// TIA Portal V16 program export: 2 tag tables, 0 data types, 2 data blocks, 14 code blocks (in call order from the OBs), 13 instance data blocks

VAR_GLOBAL   // PLC tag table "Default tag table"
   FIC_B102 AT %IW64 : Int;
   LIC_B101 AT %IW66 : Int;
   PS1_RFID_Station AT %I0.0 : Bool;   // PS-Proximity Switch
   PS2_Filling_Station AT %I0.1 : Bool;
   PS3_Quality_Station AT %I0.2 : Bool;
   PS4_End_of_Conveyor AT %I0.3 : Bool;
   T01_Low_Level AT %I0.4 : Bool;
   T01_High_Level AT %I0.5 : Bool;
   T01_Outlet AT %Q0.1 : Bool;
   T02_Outlet AT %Q0.2 : Bool;
   Outlet_Pump_Motor AT %Q0.3 : Bool;
   Conveyor_Motor AT %Q0.0 : Bool;
   NTRG_06 AT %M5.5 : Bool;
   NTRG_09 AT %M5.6 : Bool;
   NTRG_099 AT %M5.7 : Bool;
   PTRG10 AT %M6.0 : Bool;
   PTRIG999 AT %M6.1 : Bool;
   PTRIG998 AT %M6.2 : Bool;
   PTRIG888 AT %M6.3 : Bool;
   ptrig141 AT %M6.4 : Bool;
   ptrig142 AT %M6.5 : Bool;
   ptrig143 AT %M6.6 : Bool;
END_VAR

VAR_GLOBAL   // PLC tag table "P_N_TRIG"
   PTRIG1 AT %M0.0 : Bool;
   PTRIG2 AT %M0.1 : Bool;
   PTRIG3 AT %M0.2 : Bool;
   PTRIG4 AT %M0.3 : Bool;
   PTRIG5 AT %M0.4 : Bool;
   PTRIG6 AT %M0.5 : Bool;
   PTRIG7 AT %M0.6 : Bool;
   PTRIG8 AT %M0.7 : Bool;
   PTRIG9 AT %M1.0 : Bool;
   PTRIG10 AT %M1.1 : Bool;
   PTRIG11 AT %M1.2 : Bool;
   PTRIG12 AT %M1.3 : Bool;
   PTRIG13 AT %M1.4 : Bool;
   PTRIG14 AT %M1.5 : Bool;
   PTRIG15 AT %M1.6 : Bool;
   PTRIG16 AT %M1.7 : Bool;
   PTRIG17 AT %M2.0 : Bool;
   PTRIG18 AT %M2.1 : Bool;
   PTRIG19 AT %M2.2 : Bool;
   PTRIG20 AT %M2.3 : Bool;
   PTRIG21 AT %M2.4 : Bool;
   PTRIG22 AT %M2.5 : Bool;
   PTRIG23 AT %M2.6 : Bool;
   NTRIG1 AT %M2.7 : Bool;
   NTRIG2 AT %M3.0 : Bool;
   NTRIG3 AT %M3.1 : Bool;
   NTRIG4 AT %M3.2 : Bool;
   NTRIG5 AT %M3.3 : Bool;
   NTRIG6 AT %M3.4 : Bool;
   NTRIG7 AT %M3.5 : Bool;
   NTRIG8 AT %M3.6 : Bool;
   NTRIG9 AT %M3.7 : Bool;
   NTRIG10 AT %M4.0 : Bool;
   NTRIG11 AT %M4.1 : Bool;
   NTRIG12 AT %M4.2 : Bool;
   NTRIG13 AT %M4.3 : Bool;
   NTRIG14 AT %M4.4 : Bool;
   NTRIG15 AT %M4.5 : Bool;
   NTRIG16 AT %M4.6 : Bool;
   NTRIG17 AT %M4.7 : Bool;
   NTRIG18 AT %M5.0 : Bool;
   NTRIG19 AT %M5.1 : Bool;
   NTRIG20 AT %M5.2 : Bool;
   PTRIG24 AT %M5.3 : Bool;
   PTRIG25 AT %M5.4 : Bool;
END_VAR

DATA_BLOCK "DuplicateDB"   // DB12
{ S7_Optimized_Access := 'FALSE' }
VERSION : 0.1
// stored: AutoNumber true, DBAccessibleFromOPCUA true, IsOnlyStoredInLoadMemory false, IsWriteProtectedInAS false
   VAR
      Input : Struct
         FIC_B102 : Int;   // Tank2 Level Measurement
         LIC_B101 : Int;
         PS1_RFID_Station : Bool;
         PS2_Filling_Station : Bool;
         PS3_Quality_Station : Bool;
         PS4_End_of_Conveyor : Bool;
         T01_Low_Level : Bool;
         T01_High_Level : Bool;
      END_STRUCT;
   END_VAR
BEGIN
END_DATA_BLOCK

DATA_BLOCK "Global_DB"   // DB1
{ S7_Optimized_Access := 'TRUE' }
VERSION : 0.1
// stored: AutoNumber true, DBAccessibleFromOPCUA true, IsOnlyStoredInLoadMemory false, IsRetainMemResEnabled false, IsWriteProtectedInAS false, MemoryReserve 100
   VAR
      Input : Struct
         FIC_B102 : Int;   // Tank2 Level Measurement
         LIC_B101 : Int;
         PS1_RFID_Station : Bool;
         PS2_Filling_Station : Bool;
         PS3_Quality_Station : Bool;
         PS4_End_of_Conveyor : Bool;
         T01_Low_Level : Bool;
         T01_High_Level : Bool;
      END_STRUCT;
      Output : Struct
         T01_Outlet : Bool;
         T02_Outlet : Bool;
         Outlet_Pump_Motor : Bool;
         Conveyor_Motor : Bool;
         T01_Inlet : Bool;
         T02_Inlet : Bool;
      END_STRUCT;
      Other_Parameters : Struct
         Liquid_A_Filled : Bool;
         Add_Done : Bool;
         Liquid_B_Filled : Bool;
         Flow_ml_per_sec : Real;
         LiquidA_in_Bottle_ml : Real;
         LiquidB_in_Bottle_ml : Real;
         T02_Level_in_L : Real;
         T02_High_Level_Limit { ExternalVisible := 'False'} : Real;
         T02_Low_Level_Limit : Real;
         Liquid_A_pct : Int := 50;   // data from RFID tags
         Liquid_B_pct : Int := 50;   // datafrom RFID tags
         Alarm_Reset : Bool;
         operation_cycle_time : Time;
         index : Int := 1;
      END_STRUCT;
      Error : Struct
         Alarm : Word;
      END_STRUCT;
      Master_Command : Struct
         operation_begin : Bool;
         operation_finished : Bool;
      END_STRUCT;
      Production_Data : Struct   // Unit ml
         Total_Liquid_in_Bottle : Array[1..5] of Real;
         LiquidA_in_Bottle : Array[1..5] of Real;
         operation_cycles : Array[1..5] of Time;
         LiquidB_in_Bottle : Array[1..5] of Real;
         current_cycle : Int := 1;
         Bottle_Count : Int := 1;   // Total Bottle filled
      END_STRUCT;
   END_VAR
BEGIN
END_DATA_BLOCK

ORGANIZATION_BLOCK "Main"   // OB1, LAD, ProgramCycle
TITLE = "Main Program Sweep (Cycle)"
{ S7_Optimized_Access := 'TRUE' }
VERSION : 0.1
// stored: AutoNumber true, IsIECCheckEnabled false, SetENOAutomatically false
   VAR_INPUT
      Initial_Call : Bool;   // Initial call of this OB
      Remanence : Bool;   // =True, if remanent data are available
   END_VAR
   VAR_TEMP   // added for the SCL form of the ladder/FBD networks
      _w1 : Bool;
      _w2 : Bool;
   END_VAR
BEGIN

REGION Network 1: Tank 1 and Tank 2 re-filling Logic
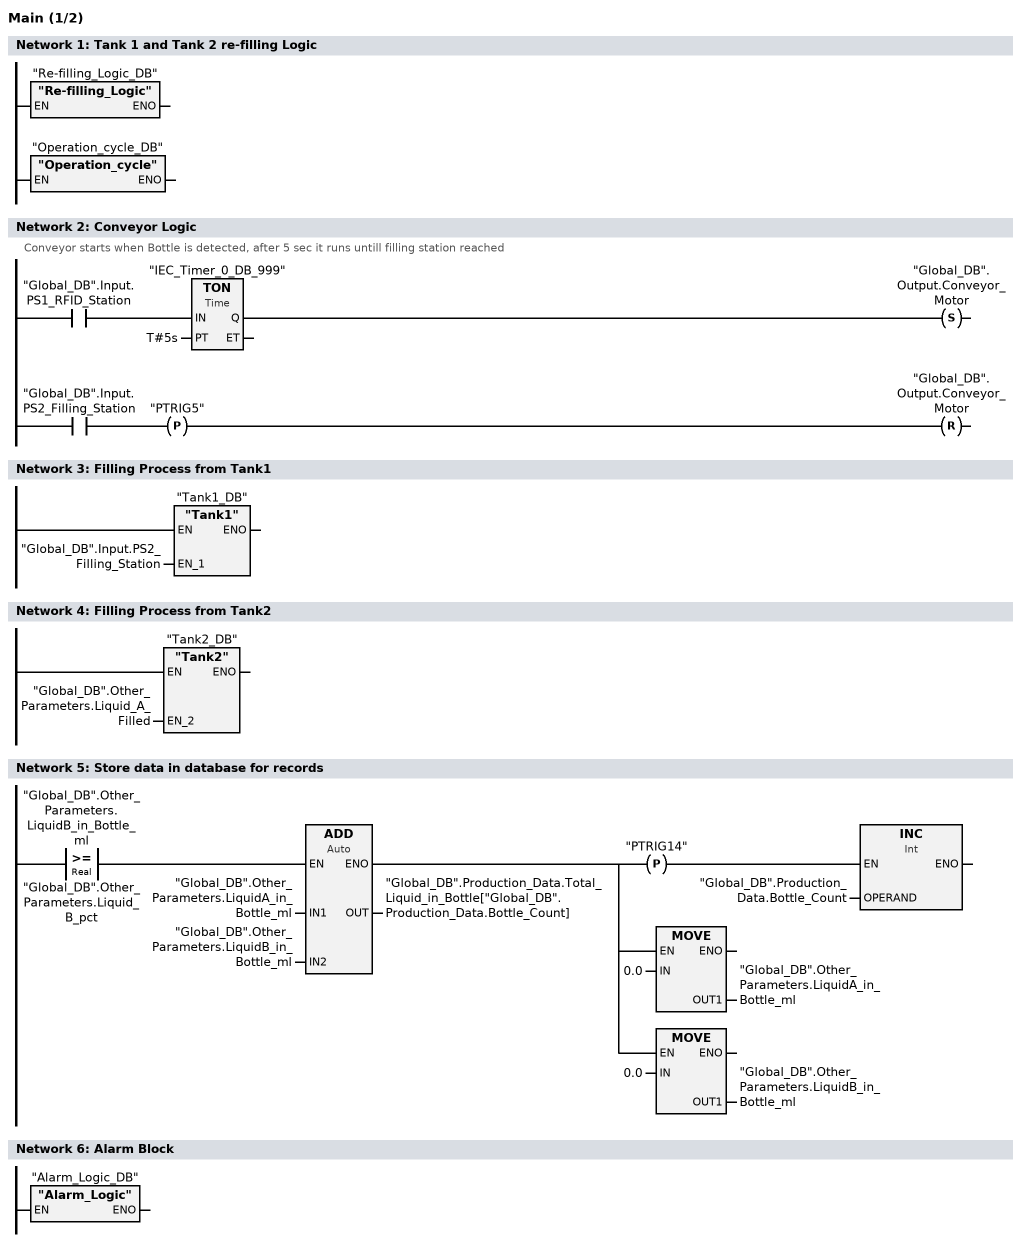
   RUNG wire#powerrail
      "Re-filling_Logic_DB"()
   END_RUNG
   RUNG wire#powerrail
      "Operation_cycle_DB"()
   END_RUNG
   // the same network as SCL:
   "Re-filling_Logic_DB"();   // "Re-filling_Logic"
   "Operation_cycle_DB"();   // "Operation_cycle"
END_REGION

REGION Network 2: Conveyor Logic
   // Conveyor starts when Bottle is detected, after 5 sec it runs untill filling station reached
   RUNG wire#powerrail
      Contact( "Global_DB".Input.PS1_RFID_Station )
      { S7_Templates := "time_type := Time" } "IEC_Timer_0_DB_999".TON(pt := T#5s, et =>)
      S_Coil( "Global_DB".Output.Conveyor_Motor )
   END_RUNG
   RUNG wire#powerrail
      Contact( "Global_DB".Input.PS2_Filling_Station )
      P_Trig( "PTRIG5" )
      R_Coil( "Global_DB".Output.Conveyor_Motor )
   END_RUNG
   // the same network as SCL:
   "IEC_Timer_0_DB_999".TON(IN := "Global_DB".Input.PS1_RFID_Station, PT := T#5s);
   IF "IEC_Timer_0_DB_999".Q THEN "Global_DB".Output.Conveyor_Motor := TRUE; END_IF;
   #_w1 := "Global_DB".Input.PS2_Filling_Station AND NOT "PTRIG5";   // rising edge
   "PTRIG5" := "Global_DB".Input.PS2_Filling_Station;
   IF #_w1 THEN "Global_DB".Output.Conveyor_Motor := FALSE; END_IF;
END_REGION

REGION Network 3: Filling Process from Tank1
   RUNG wire#powerrail
      "Tank1_DB"(EN_1 := "Global_DB".Input.PS2_Filling_Station)
   END_RUNG
   // the same network as SCL:
   "Tank1_DB"(EN_1 := "Global_DB".Input.PS2_Filling_Station);   // "Tank1"
END_REGION

REGION Network 4: Filling Process from Tank2
   RUNG wire#powerrail
      "Tank2_DB"(EN_2 := "Global_DB".Other_Parameters.Liquid_A_Filled)
   END_RUNG
   // the same network as SCL:
   "Tank2_DB"(EN_2 := "Global_DB".Other_Parameters.Liquid_A_Filled);   // "Tank2"
END_REGION

REGION Network 5: Store data in database for records
   RUNG wire#powerrail
      { S7_Templates := "SrcType := Real" } GE_Contact(in1 := "Global_DB".Other_Parameters.LiquidB_in_Bottle_ml, in2 := "Global_DB".Other_Parameters.Liquid_B_pct)
      Add(in1 := "Global_DB".Other_Parameters.LiquidA_in_Bottle_ml, in2 := "Global_DB".Other_Parameters.LiquidB_in_Bottle_ml, out => "Global_DB".Production_Data.Total_Liquid_in_Bottle["Global_DB".Production_Data.Bottle_Count])
      wire#w1
      P_Trig( "PTRIG14" )
      { S7_Templates := "DestType := Int" } Inc( "Global_DB".Production_Data.Bottle_Count )
   END_RUNG
   RUNG wire#w1
      Move(in := 0.0, out1 => "Global_DB".Other_Parameters.LiquidA_in_Bottle_ml)
   END_RUNG
   RUNG wire#w1
      Move(in := 0.0, out1 => "Global_DB".Other_Parameters.LiquidB_in_Bottle_ml)
   END_RUNG
   // the same network as SCL:
   #_w1 := "Global_DB".Other_Parameters.LiquidB_in_Bottle_ml >= "Global_DB".Other_Parameters.Liquid_B_pct;
   IF #_w1 THEN
       "Global_DB".Production_Data.Total_Liquid_in_Bottle["Global_DB".Production_Data.Bottle_Count] := "Global_DB".Other_Parameters.LiquidA_in_Bottle_ml + "Global_DB".Other_Parameters.LiquidB_in_Bottle_ml;
   END_IF;
   #_w2 := #_w1 AND NOT "PTRIG14";   // rising edge
   "PTRIG14" := #_w1;
   IF #_w2 THEN
       "Global_DB".Production_Data.Bottle_Count := "Global_DB".Production_Data.Bottle_Count + 1;
   END_IF;
   IF #_w1 THEN
       "Global_DB".Other_Parameters.LiquidA_in_Bottle_ml := 0.0;
       "Global_DB".Other_Parameters.LiquidB_in_Bottle_ml := 0.0;
   END_IF;
END_REGION

REGION Network 6: Alarm Block
   RUNG wire#powerrail
      "Alarm_Logic_DB"()
   END_RUNG
   // the same network as SCL:
   "Alarm_Logic_DB"();   // "Alarm_Logic"
END_REGION

REGION Network 7: Process after bottle is filled
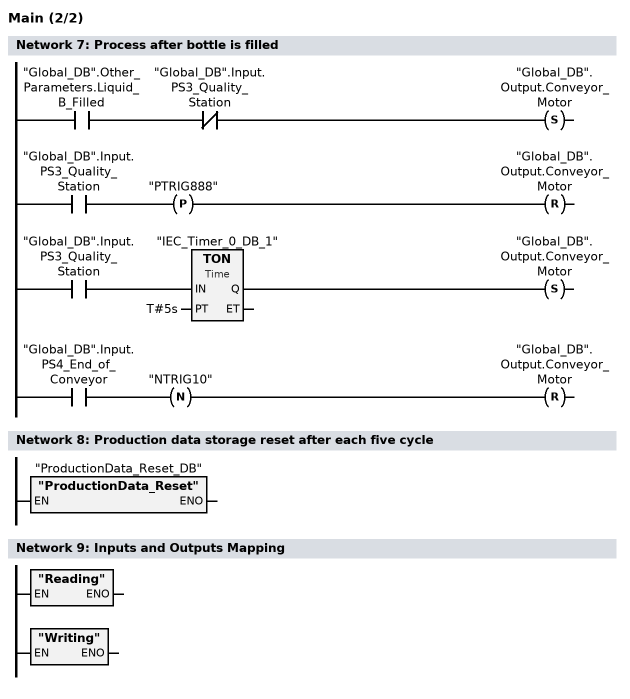
   RUNG wire#powerrail
      Contact( "Global_DB".Other_Parameters.Liquid_B_Filled )
      I_Contact( "Global_DB".Input.PS3_Quality_Station )
      S_Coil( "Global_DB".Output.Conveyor_Motor )
   END_RUNG
   RUNG wire#powerrail
      Contact( "Global_DB".Input.PS3_Quality_Station )
      P_Trig( "PTRIG888" )
      R_Coil( "Global_DB".Output.Conveyor_Motor )
   END_RUNG
   RUNG wire#powerrail
      Contact( "Global_DB".Input.PS3_Quality_Station )
      { S7_Templates := "time_type := Time" } "IEC_Timer_0_DB_1".TON(pt := T#5s, et =>)
      S_Coil( "Global_DB".Output.Conveyor_Motor )
   END_RUNG
   RUNG wire#powerrail
      Contact( "Global_DB".Input.PS4_End_of_Conveyor )
      N_Trig( "NTRIG10" )
      R_Coil( "Global_DB".Output.Conveyor_Motor )
   END_RUNG
   // the same network as SCL:
   IF "Global_DB".Other_Parameters.Liquid_B_Filled AND NOT "Global_DB".Input.PS3_Quality_Station THEN
       "Global_DB".Output.Conveyor_Motor := TRUE;
   END_IF;
   #_w1 := "Global_DB".Input.PS3_Quality_Station AND NOT "PTRIG888";   // rising edge
   "PTRIG888" := "Global_DB".Input.PS3_Quality_Station;
   IF #_w1 THEN "Global_DB".Output.Conveyor_Motor := FALSE; END_IF;
   "IEC_Timer_0_DB_1".TON(IN := "Global_DB".Input.PS3_Quality_Station, PT := T#5s);
   IF "IEC_Timer_0_DB_1".Q THEN "Global_DB".Output.Conveyor_Motor := TRUE; END_IF;
   #_w2 := NOT "Global_DB".Input.PS4_End_of_Conveyor AND "NTRIG10";   // falling edge
   "NTRIG10" := "Global_DB".Input.PS4_End_of_Conveyor;
   IF #_w2 THEN "Global_DB".Output.Conveyor_Motor := FALSE; END_IF;
END_REGION

REGION Network 8: Production data storage reset after each five cycle
   RUNG wire#powerrail
      "ProductionData_Reset_DB"()
   END_RUNG
   // the same network as SCL:
   "ProductionData_Reset_DB"();   // "ProductionData_Reset"
END_REGION

REGION Network 9: Inputs and Outputs Mapping
   RUNG wire#powerrail
      "Reading"()
   END_RUNG
   RUNG wire#powerrail
      "Writing"()
   END_RUNG
   // the same network as SCL:
   "Reading"();
   "Writing"();
END_REGION
END_ORGANIZATION_BLOCK

FUNCTION_BLOCK "Re-filling_Logic"   // FB1, LAD
{ S7_Optimized_Access := 'TRUE' }
VERSION : 0.1
// stored: AutoNumber true, IsIECCheckEnabled false, IsRetainMemResEnabled false, MemoryReserve 100, SetENOAutomatically false, UDAEnableTagReadback false
   VAR_TEMP   // added for the SCL form of the ladder/FBD networks
      _w1 : Bool;
      _w2 : Bool;
      _w3 : Bool;
      _w4 : Bool;
   END_VAR
BEGIN

REGION Network 1: Tank2 Re-filling Proccess
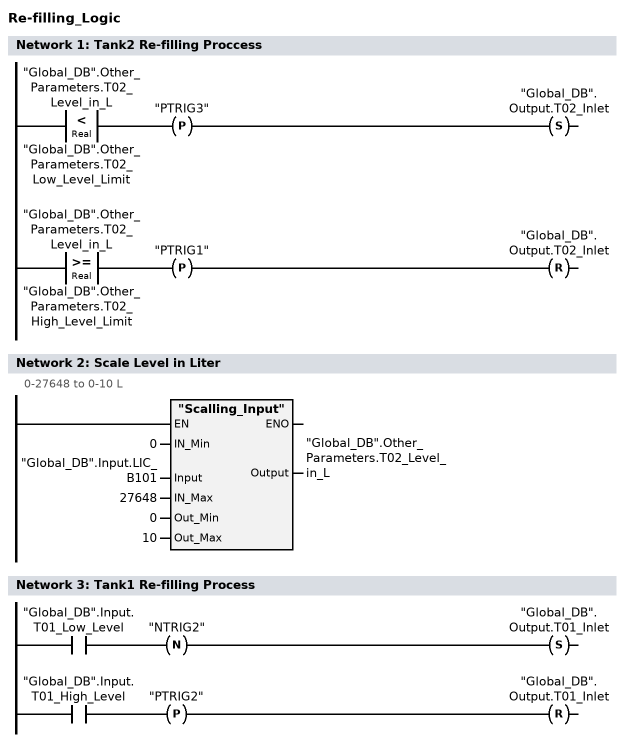
   RUNG wire#powerrail
      { S7_Templates := "SrcType := Real" } LT_Contact(in1 := "Global_DB".Other_Parameters.T02_Level_in_L, in2 := "Global_DB".Other_Parameters.T02_Low_Level_Limit)
      P_Trig( "PTRIG3" )
      S_Coil( "Global_DB".Output.T02_Inlet )
   END_RUNG
   RUNG wire#powerrail
      { S7_Templates := "SrcType := Real" } GE_Contact(in1 := "Global_DB".Other_Parameters.T02_Level_in_L, in2 := "Global_DB".Other_Parameters.T02_High_Level_Limit)
      P_Trig( "PTRIG1" )
      R_Coil( "Global_DB".Output.T02_Inlet )
   END_RUNG
   // the same network as SCL:
   #_w1 := "Global_DB".Other_Parameters.T02_Level_in_L < "Global_DB".Other_Parameters.T02_Low_Level_Limit;
   #_w2 := #_w1 AND NOT "PTRIG3";   // rising edge
   "PTRIG3" := #_w1;
   IF #_w2 THEN "Global_DB".Output.T02_Inlet := TRUE; END_IF;
   #_w3 := "Global_DB".Other_Parameters.T02_Level_in_L >= "Global_DB".Other_Parameters.T02_High_Level_Limit;
   #_w4 := #_w3 AND NOT "PTRIG1";   // rising edge
   "PTRIG1" := #_w3;
   IF #_w4 THEN "Global_DB".Output.T02_Inlet := FALSE; END_IF;
END_REGION

REGION Network 2: Scale Level in Liter
   // 0-27648 to 0-10 L
   RUNG wire#powerrail
      "Scalling_Input"(IN_Min := 0, Input := "Global_DB".Input.LIC_B101, IN_Max := 27648, Out_Min := 0, Out_Max := 10, Output => "Global_DB".Other_Parameters.T02_Level_in_L)
   END_RUNG
   // the same network as SCL:
   "Scalling_Input"(IN_Min := 0,
                    Input := "Global_DB".Input.LIC_B101,
                    IN_Max := 27648,
                    Out_Min := 0,
                    Out_Max := 10,
                    Output => "Global_DB".Other_Parameters.T02_Level_in_L);
END_REGION

REGION Network 3: Tank1 Re-filling Process
   RUNG wire#powerrail
      Contact( "Global_DB".Input.T01_Low_Level )
      N_Trig( "NTRIG2" )
      S_Coil( "Global_DB".Output.T01_Inlet )
   END_RUNG
   RUNG wire#powerrail
      Contact( "Global_DB".Input.T01_High_Level )
      P_Trig( "PTRIG2" )
      R_Coil( "Global_DB".Output.T01_Inlet )
   END_RUNG
   // the same network as SCL:
   #_w1 := NOT "Global_DB".Input.T01_Low_Level AND "NTRIG2";   // falling edge
   "NTRIG2" := "Global_DB".Input.T01_Low_Level;
   IF #_w1 THEN "Global_DB".Output.T01_Inlet := TRUE; END_IF;
   #_w2 := "Global_DB".Input.T01_High_Level AND NOT "PTRIG2";   // rising edge
   "PTRIG2" := "Global_DB".Input.T01_High_Level;
   IF #_w2 THEN "Global_DB".Output.T01_Inlet := FALSE; END_IF;
END_REGION
END_FUNCTION_BLOCK

FUNCTION "Scalling_Input" : Void   // FC1, FBD
{ S7_Optimized_Access := 'TRUE' }
VERSION : 0.1
// stored: AutoNumber true, IsIECCheckEnabled false, SetENOAutomatically false, UDAEnableTagReadback false
   VAR_INPUT
      IN_Min : Int;
      Input : Int;
      IN_Max : Int;
      Out_Min : Int;
      Out_Max : Int;
   END_VAR
   VAR_OUTPUT
      Output : Real;
   END_VAR
   VAR_TEMP
      Normed : Real;
   END_VAR
BEGIN

REGION Network 1
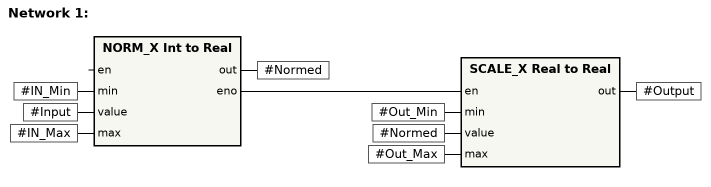
   #Normed := NORM_X(MIN := #IN_Min, VALUE := #Input, MAX := #IN_Max);
   #Output := SCALE_X(MIN := #Out_Min, VALUE := #Normed, MAX := #Out_Max);
END_REGION
END_FUNCTION

FUNCTION_BLOCK "Operation_cycle"   // FB8, LAD
{ S7_Optimized_Access := 'TRUE' }
VERSION : 0.1
// stored: AutoNumber true, IsIECCheckEnabled false, IsRetainMemResEnabled false, MemoryReserve 100, SetENOAutomatically false, UDAEnableTagReadback false
   VAR
      begun : Bool;
   END_VAR
   VAR_TEMP   // added for the SCL form of the ladder/FBD networks
      _w1 : Bool;
      _w2 : Bool;
      _w3 : Bool;
   END_VAR
BEGIN

REGION Network 1
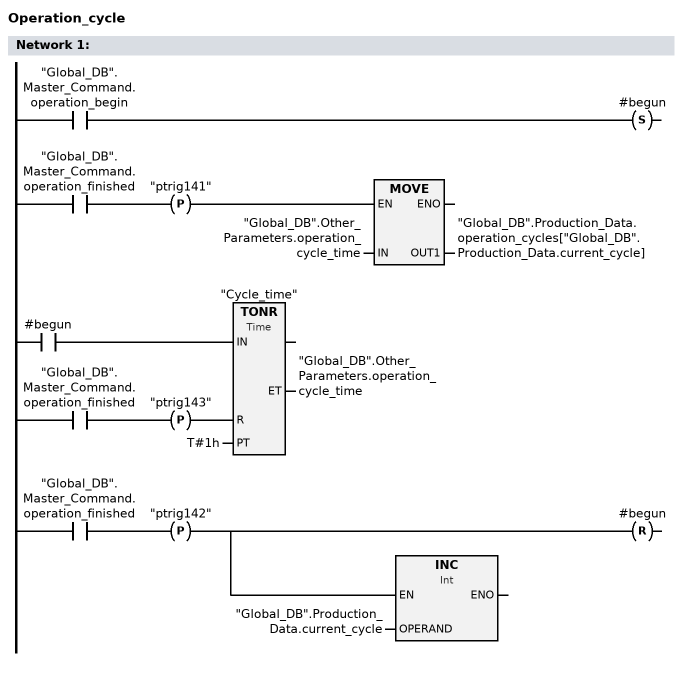
   RUNG wire#powerrail
      Contact( "Global_DB".Master_Command.operation_begin )
      S_Coil( #begun )
   END_RUNG
   RUNG wire#powerrail
      Contact( "Global_DB".Master_Command.operation_finished )
      P_Trig( "ptrig141" )
      Move(in := "Global_DB".Other_Parameters.operation_cycle_time, out1 => "Global_DB".Production_Data.operation_cycles["Global_DB".Production_Data.current_cycle])
   END_RUNG
   RUNG wire#powerrail
      Contact( #begun )
      { S7_Templates := "time_type := Time" } "Cycle_time".TONR(r := wire#w1, pt := T#1h, et => "Global_DB".Other_Parameters.operation_cycle_time)
   END_RUNG
   RUNG wire#powerrail
      Contact( "Global_DB".Master_Command.operation_finished )
      P_Trig( "ptrig143" )
   END_RUNG wire#w1
   RUNG wire#powerrail
      Contact( "Global_DB".Master_Command.operation_finished )
      P_Trig( "ptrig142" )
      wire#w2
      R_Coil( #begun )
   END_RUNG
   RUNG wire#w2
      { S7_Templates := "DestType := Int" } Inc( "Global_DB".Production_Data.current_cycle )
   END_RUNG
   // the same network as SCL:
   IF "Global_DB".Master_Command.operation_begin THEN #begun := TRUE; END_IF;
   #_w1 := "Global_DB".Master_Command.operation_finished AND NOT "ptrig141";   // rising edge
   "ptrig141" := "Global_DB".Master_Command.operation_finished;
   IF #_w1 THEN
       "Global_DB".Production_Data.operation_cycles["Global_DB".Production_Data.current_cycle] := "Global_DB".Other_Parameters.operation_cycle_time;
   END_IF;
   #_w2 := "Global_DB".Master_Command.operation_finished AND NOT "ptrig143";   // rising edge
   "ptrig143" := "Global_DB".Master_Command.operation_finished;
   "Cycle_time".TONR(IN := #begun,
                     R := #_w2,
                     PT := T#1h,
                     ET => "Global_DB".Other_Parameters.operation_cycle_time);
   #_w3 := "Global_DB".Master_Command.operation_finished AND NOT "ptrig142";   // rising edge
   "ptrig142" := "Global_DB".Master_Command.operation_finished;
   IF #_w3 THEN
       #begun := FALSE;
       "Global_DB".Production_Data.current_cycle := "Global_DB".Production_Data.current_cycle + 1;
   END_IF;
END_REGION
END_FUNCTION_BLOCK

FUNCTION_BLOCK "Tank1"   // FB4, LAD
{ S7_Optimized_Access := 'TRUE' }
VERSION : 0.1
// stored: AutoNumber true, IsIECCheckEnabled false, IsRetainMemResEnabled false, MemoryReserve 100, SetENOAutomatically false, UDAEnableTagReadback false
   VAR_INPUT
      EN_1 : Bool;
   END_VAR
   VAR_TEMP   // added for the SCL form of the ladder/FBD networks
      _w1 : Bool;
      _w2 : Bool;
      _w3 : Bool;
   END_VAR
BEGIN

REGION Network 1: Filling Process from Tank1
   // 0-27648 to 0-250ml
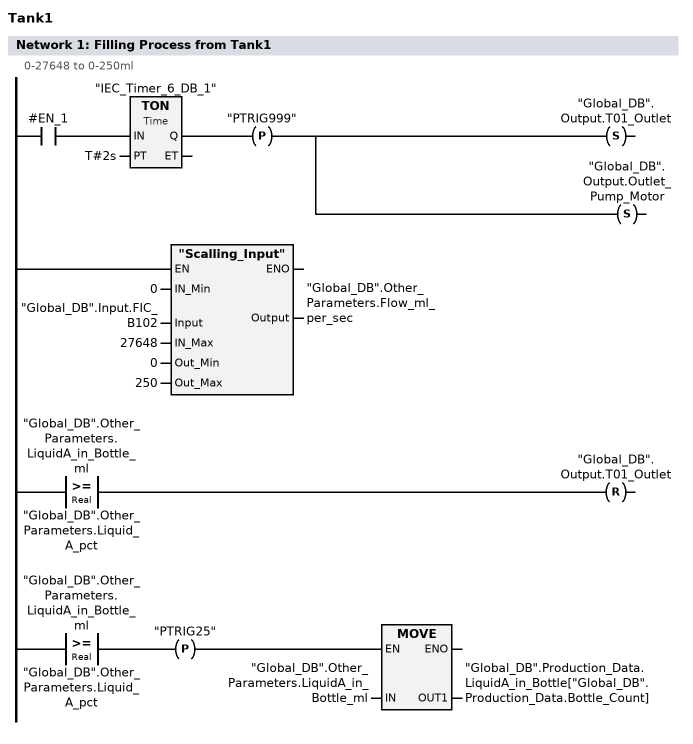
   RUNG wire#powerrail
      Contact( #EN_1 )
      { S7_Templates := "time_type := Time" } "IEC_Timer_6_DB_1".TON(pt := T#2s, et =>)
      P_Trig( "PTRIG999" )
      wire#w1
      S_Coil( "Global_DB".Output.T01_Outlet )
   END_RUNG
   RUNG wire#w1
      S_Coil( "Global_DB".Output.Outlet_Pump_Motor )
   END_RUNG
   RUNG wire#powerrail
      "Scalling_Input"(IN_Min := 0, Input := "Global_DB".Input.FIC_B102, IN_Max := 27648, Out_Min := 0, Out_Max := 250, Output => "Global_DB".Other_Parameters.Flow_ml_per_sec)
   END_RUNG
   RUNG wire#powerrail
      { S7_Templates := "SrcType := Real" } GE_Contact(in1 := "Global_DB".Other_Parameters.LiquidA_in_Bottle_ml, in2 := "Global_DB".Other_Parameters.Liquid_A_pct)
      R_Coil( "Global_DB".Output.T01_Outlet )
   END_RUNG
   RUNG wire#powerrail
      { S7_Templates := "SrcType := Real" } GE_Contact(in1 := "Global_DB".Other_Parameters.LiquidA_in_Bottle_ml, in2 := "Global_DB".Other_Parameters.Liquid_A_pct)
      P_Trig( "PTRIG25" )
      Move(in := "Global_DB".Other_Parameters.LiquidA_in_Bottle_ml, out1 => "Global_DB".Production_Data.LiquidA_in_Bottle["Global_DB".Production_Data.Bottle_Count])
   END_RUNG
   // the same network as SCL:
   "IEC_Timer_6_DB_1".TON(IN := #EN_1, PT := T#2s);
   #_w1 := "IEC_Timer_6_DB_1".Q AND NOT "PTRIG999";   // rising edge
   "PTRIG999" := "IEC_Timer_6_DB_1".Q;
   IF #_w1 THEN
       "Global_DB".Output.T01_Outlet := TRUE;
       "Global_DB".Output.Outlet_Pump_Motor := TRUE;
   END_IF;
   "Scalling_Input"(IN_Min := 0,
                    Input := "Global_DB".Input.FIC_B102,
                    IN_Max := 27648,
                    Out_Min := 0,
                    Out_Max := 250,
                    Output => "Global_DB".Other_Parameters.Flow_ml_per_sec);
   IF "Global_DB".Other_Parameters.LiquidA_in_Bottle_ml >= "Global_DB".Other_Parameters.Liquid_A_pct THEN
       "Global_DB".Output.T01_Outlet := FALSE;
   END_IF;
   #_w2 := "Global_DB".Other_Parameters.LiquidA_in_Bottle_ml >= "Global_DB".Other_Parameters.Liquid_A_pct;
   #_w3 := #_w2 AND NOT "PTRIG25";   // rising edge
   "PTRIG25" := #_w2;
   IF #_w3 THEN
       "Global_DB".Production_Data.LiquidA_in_Bottle["Global_DB".Production_Data.Bottle_Count] := "Global_DB".Other_Parameters.LiquidA_in_Bottle_ml;
   END_IF;
END_REGION
END_FUNCTION_BLOCK

FUNCTION_BLOCK "Tank2"   // FB5, LAD
{ S7_Optimized_Access := 'TRUE' }
VERSION : 0.1
// stored: AutoNumber true, IsIECCheckEnabled false, IsRetainMemResEnabled false, MemoryReserve 100, SetENOAutomatically false, UDAEnableTagReadback false
   VAR_INPUT
      EN_2 : Bool;
   END_VAR
   VAR_TEMP   // added for the SCL form of the ladder/FBD networks
      _w1 : Bool;
      _w2 : Bool;
      _w3 : Bool;
   END_VAR
BEGIN

REGION Network 1
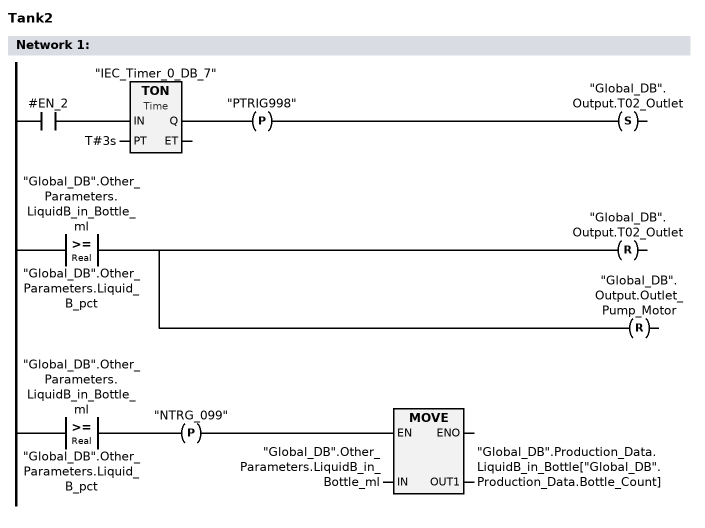
   RUNG wire#powerrail
      Contact( #EN_2 )
      { S7_Templates := "time_type := Time" } "IEC_Timer_0_DB_7".TON(pt := T#3s, et =>)
      P_Trig( "PTRIG998" )
      S_Coil( "Global_DB".Output.T02_Outlet )
   END_RUNG
   RUNG wire#powerrail
      { S7_Templates := "SrcType := Real" } GE_Contact(in1 := "Global_DB".Other_Parameters.LiquidB_in_Bottle_ml, in2 := "Global_DB".Other_Parameters.Liquid_B_pct)
      wire#w1
      R_Coil( "Global_DB".Output.T02_Outlet )
   END_RUNG
   RUNG wire#w1
      R_Coil( "Global_DB".Output.Outlet_Pump_Motor )
   END_RUNG
   RUNG wire#powerrail
      { S7_Templates := "SrcType := Real" } GE_Contact(in1 := "Global_DB".Other_Parameters.LiquidB_in_Bottle_ml, in2 := "Global_DB".Other_Parameters.Liquid_B_pct)
      P_Trig( "NTRG_099" )
      Move(in := "Global_DB".Other_Parameters.LiquidB_in_Bottle_ml, out1 => "Global_DB".Production_Data.LiquidB_in_Bottle["Global_DB".Production_Data.Bottle_Count])
   END_RUNG
   // the same network as SCL:
   "IEC_Timer_0_DB_7".TON(IN := #EN_2, PT := T#3s);
   #_w1 := "IEC_Timer_0_DB_7".Q AND NOT "PTRIG998";   // rising edge
   "PTRIG998" := "IEC_Timer_0_DB_7".Q;
   IF #_w1 THEN "Global_DB".Output.T02_Outlet := TRUE; END_IF;
   IF "Global_DB".Other_Parameters.LiquidB_in_Bottle_ml >= "Global_DB".Other_Parameters.Liquid_B_pct THEN
       "Global_DB".Output.T02_Outlet := FALSE;
       "Global_DB".Output.Outlet_Pump_Motor := FALSE;
   END_IF;
   #_w2 := "Global_DB".Other_Parameters.LiquidB_in_Bottle_ml >= "Global_DB".Other_Parameters.Liquid_B_pct;
   #_w3 := #_w2 AND NOT "NTRG_099";   // rising edge
   "NTRG_099" := #_w2;
   IF #_w3 THEN
       "Global_DB".Production_Data.LiquidB_in_Bottle["Global_DB".Production_Data.Bottle_Count] := "Global_DB".Other_Parameters.LiquidB_in_Bottle_ml;
   END_IF;
END_REGION
END_FUNCTION_BLOCK

FUNCTION_BLOCK "Alarm_Logic"   // FB3, LAD
{ S7_Optimized_Access := 'TRUE' }
VERSION : 0.1
// stored: AutoNumber true, IsIECCheckEnabled false, IsRetainMemResEnabled false, MemoryReserve 100, SetENOAutomatically false, UDAEnableTagReadback false
   VAR_TEMP   // added for the SCL form of the ladder/FBD networks
      _w1 : Bool;
      _w2 : Bool;
      _w3 : Bool;
      _w4 : Bool;
      _w5 : Bool;
      _w6 : Bool;
   END_VAR
BEGIN

REGION Network 1: Bottle Overfilled Alarm
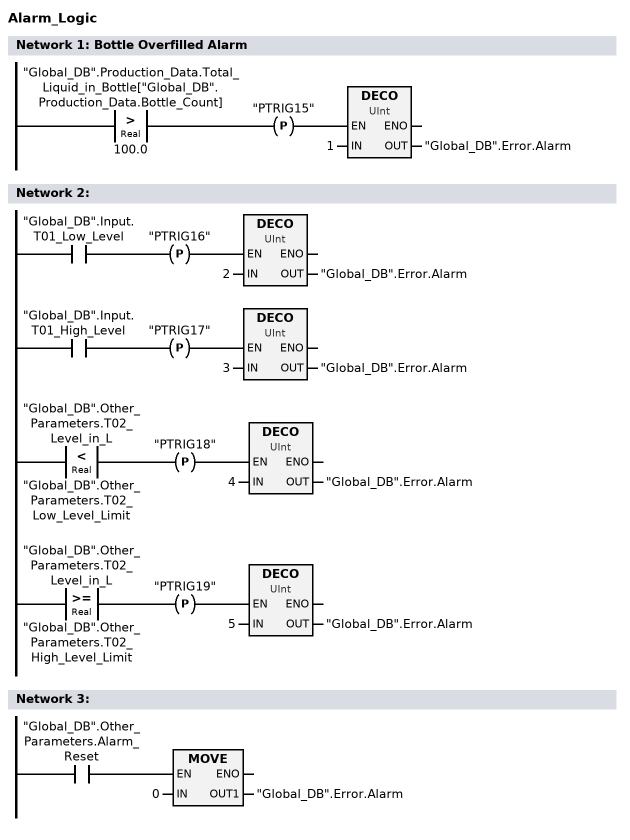
   RUNG wire#powerrail
      { S7_Templates := "SrcType := Real" } GT_Contact(in1 := "Global_DB".Production_Data.Total_Liquid_in_Bottle["Global_DB".Production_Data.Bottle_Count], in2 := 100.0)
      P_Trig( "PTRIG15" )
      { S7_Templates := "[value_type := UInt, return_type := Word]" } DECO(IN := 1, OUT => "Global_DB".Error.Alarm)
   END_RUNG
   // the same network as SCL:
   #_w1 := "Global_DB".Production_Data.Total_Liquid_in_Bottle["Global_DB".Production_Data.Bottle_Count] > 100.0;
   #_w2 := #_w1 AND NOT "PTRIG15";   // rising edge
   "PTRIG15" := #_w1;
   IF #_w2 THEN DECO(IN := 1, OUT => "Global_DB".Error.Alarm); END_IF;
END_REGION

REGION Network 2
   RUNG wire#powerrail
      Contact( "Global_DB".Input.T01_Low_Level )
      P_Trig( "PTRIG16" )
      { S7_Templates := "[value_type := UInt, return_type := Word]" } DECO(IN := 2, OUT => "Global_DB".Error.Alarm)
   END_RUNG
   RUNG wire#powerrail
      Contact( "Global_DB".Input.T01_High_Level )
      P_Trig( "PTRIG17" )
      { S7_Templates := "[value_type := UInt, return_type := Word]" } DECO(IN := 3, OUT => "Global_DB".Error.Alarm)
   END_RUNG
   RUNG wire#powerrail
      { S7_Templates := "SrcType := Real" } LT_Contact(in1 := "Global_DB".Other_Parameters.T02_Level_in_L, in2 := "Global_DB".Other_Parameters.T02_Low_Level_Limit)
      P_Trig( "PTRIG18" )
      { S7_Templates := "[value_type := UInt, return_type := Word]" } DECO(IN := 4, OUT => "Global_DB".Error.Alarm)
   END_RUNG
   RUNG wire#powerrail
      { S7_Templates := "SrcType := Real" } GE_Contact(in1 := "Global_DB".Other_Parameters.T02_Level_in_L, in2 := "Global_DB".Other_Parameters.T02_High_Level_Limit)
      P_Trig( "PTRIG19" )
      { S7_Templates := "[value_type := UInt, return_type := Word]" } DECO(IN := 5, OUT => "Global_DB".Error.Alarm)
   END_RUNG
   // the same network as SCL:
   #_w1 := "Global_DB".Input.T01_Low_Level AND NOT "PTRIG16";   // rising edge
   "PTRIG16" := "Global_DB".Input.T01_Low_Level;
   IF #_w1 THEN DECO(IN := 2, OUT => "Global_DB".Error.Alarm); END_IF;
   #_w2 := "Global_DB".Input.T01_High_Level AND NOT "PTRIG17";   // rising edge
   "PTRIG17" := "Global_DB".Input.T01_High_Level;
   IF #_w2 THEN DECO(IN := 3, OUT => "Global_DB".Error.Alarm); END_IF;
   #_w3 := "Global_DB".Other_Parameters.T02_Level_in_L < "Global_DB".Other_Parameters.T02_Low_Level_Limit;
   #_w4 := #_w3 AND NOT "PTRIG18";   // rising edge
   "PTRIG18" := #_w3;
   IF #_w4 THEN DECO(IN := 4, OUT => "Global_DB".Error.Alarm); END_IF;
   #_w5 := "Global_DB".Other_Parameters.T02_Level_in_L >= "Global_DB".Other_Parameters.T02_High_Level_Limit;
   #_w6 := #_w5 AND NOT "PTRIG19";   // rising edge
   "PTRIG19" := #_w5;
   IF #_w6 THEN DECO(IN := 5, OUT => "Global_DB".Error.Alarm); END_IF;
END_REGION

REGION Network 3
   RUNG wire#powerrail
      Contact( "Global_DB".Other_Parameters.Alarm_Reset )
      Move(in := 0, out1 => "Global_DB".Error.Alarm)
   END_RUNG
   // the same network as SCL:
   IF "Global_DB".Other_Parameters.Alarm_Reset THEN "Global_DB".Error.Alarm := 0; END_IF;
END_REGION
END_FUNCTION_BLOCK

FUNCTION_BLOCK "ProductionData_Reset"
{ S7_Optimized_Access := 'TRUE' }
VERSION : 0.1

BEGIN
	IF "Global_DB".Production_Data.Bottle_Count > 5 THEN
	    FOR "Global_DB".Other_Parameters.index := 1 TO 5 BY 1 DO
	        "Global_DB".Production_Data.Total_Liquid_in_Bottle["Global_DB".Other_Parameters.index] := 0.0;
	        "Global_DB".Production_Data.LiquidA_in_Bottle["Global_DB".Other_Parameters.index] := 0.0;
	        "Global_DB".Production_Data.LiquidB_in_Bottle["Global_DB".Other_Parameters.index] := 0.0;
	    END_FOR;
	    
	    "Global_DB".Production_Data.Bottle_Count := 1;
	    
	 END_IF;
	
END_FUNCTION_BLOCK

FUNCTION "Reading" : Void
{ S7_Optimized_Access := 'TRUE' }
VERSION : 0.1

BEGIN
	// Reading inputs from PLC terminals to Global_DB
	
	"Global_DB".Input.FIC_B102 := "FIC_B102";
	"Global_DB".Input.LIC_B101 := "LIC_B101";
	"Global_DB".Input.PS1_RFID_Station := "PS1_RFID_Station";
	"Global_DB".Input.PS2_Filling_Station := "PS2_Filling_Station";
	"Global_DB".Input.PS3_Quality_Station := "PS3_Quality_Station";
	"Global_DB".Input.PS4_End_of_Conveyor := "PS4_End_of_Conveyor";
	"Global_DB".Input.T01_Low_Level := "T01_Low_Level";
	"Global_DB".Input.T01_High_Level := "T01_High_Level";
	
END_FUNCTION

FUNCTION "Writing" : Void
{ S7_Optimized_Access := 'TRUE' }
VERSION : 0.1

BEGIN
	// Writing Output from Global_DB to PLC Terminal
	
	"T01_Outlet" := "Global_DB".Output.T01_Outlet;
	"T02_Outlet" := "Global_DB".Output.T02_Outlet;
	
	"Outlet_Pump_Motor" := "Global_DB".Output.Outlet_Pump_Motor;
	"Conveyor_Motor" := "Global_DB".Output.Conveyor_Motor;
END_FUNCTION

ORGANIZATION_BLOCK "Totalizer"   // OB30, LAD, CyclicInterrupt
{ S7_Optimized_Access := 'TRUE' }
VERSION : 0.1
// stored: AutoNumber true, IsIECCheckEnabled false, SetENOAutomatically false
   VAR_INPUT
      Initial_Call : Bool;   // Initial call of this OB
      Event_Count : Int;   // Events discarded
   END_VAR
BEGIN

REGION Network 1: Tank1 - LiquidA filling value Totalizer
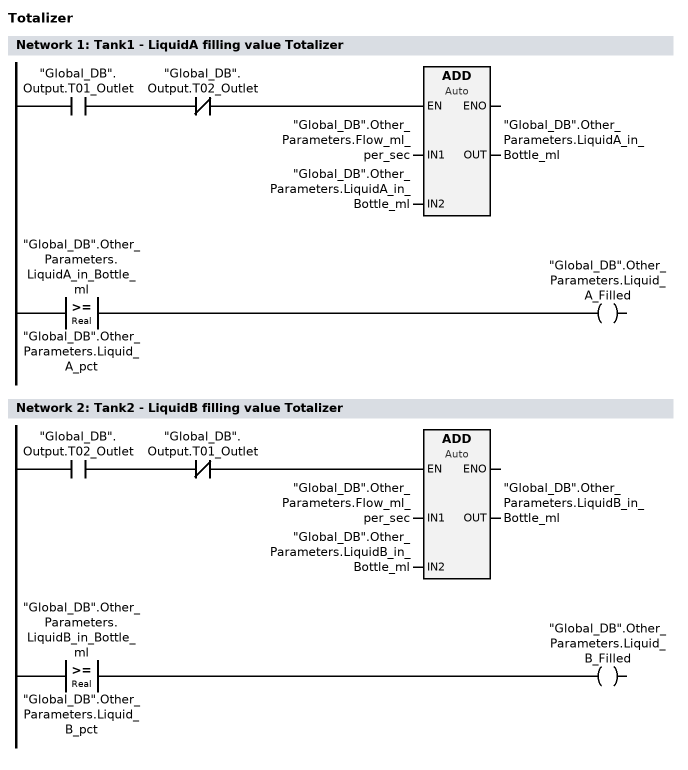
   RUNG wire#powerrail
      Contact( "Global_DB".Output.T01_Outlet )
      I_Contact( "Global_DB".Output.T02_Outlet )
      Add(in1 := "Global_DB".Other_Parameters.Flow_ml_per_sec, in2 := "Global_DB".Other_Parameters.LiquidA_in_Bottle_ml, out => "Global_DB".Other_Parameters.LiquidA_in_Bottle_ml)
   END_RUNG
   RUNG wire#powerrail
      { S7_Templates := "SrcType := Real" } GE_Contact(in1 := "Global_DB".Other_Parameters.LiquidA_in_Bottle_ml, in2 := "Global_DB".Other_Parameters.Liquid_A_pct)
      Coil( "Global_DB".Other_Parameters.Liquid_A_Filled )
   END_RUNG
   // the same network as SCL:
   IF "Global_DB".Output.T01_Outlet AND NOT "Global_DB".Output.T02_Outlet THEN
       "Global_DB".Other_Parameters.LiquidA_in_Bottle_ml := "Global_DB".Other_Parameters.Flow_ml_per_sec + "Global_DB".Other_Parameters.LiquidA_in_Bottle_ml;
   END_IF;
   "Global_DB".Other_Parameters.Liquid_A_Filled := "Global_DB".Other_Parameters.LiquidA_in_Bottle_ml >= "Global_DB".Other_Parameters.Liquid_A_pct;
END_REGION

REGION Network 2: Tank2 - LiquidB filling value Totalizer
   RUNG wire#powerrail
      Contact( "Global_DB".Output.T02_Outlet )
      I_Contact( "Global_DB".Output.T01_Outlet )
      Add(in1 := "Global_DB".Other_Parameters.Flow_ml_per_sec, in2 := "Global_DB".Other_Parameters.LiquidB_in_Bottle_ml, out => "Global_DB".Other_Parameters.LiquidB_in_Bottle_ml)
   END_RUNG
   RUNG wire#powerrail
      { S7_Templates := "SrcType := Real" } GE_Contact(in1 := "Global_DB".Other_Parameters.LiquidB_in_Bottle_ml, in2 := "Global_DB".Other_Parameters.Liquid_B_pct)
      Coil( "Global_DB".Other_Parameters.Liquid_B_Filled )
   END_RUNG
   // the same network as SCL:
   IF "Global_DB".Output.T02_Outlet AND NOT "Global_DB".Output.T01_Outlet THEN
       "Global_DB".Other_Parameters.LiquidB_in_Bottle_ml := "Global_DB".Other_Parameters.Flow_ml_per_sec + "Global_DB".Other_Parameters.LiquidB_in_Bottle_ml;
   END_IF;
   "Global_DB".Other_Parameters.Liquid_B_Filled := "Global_DB".Other_Parameters.LiquidB_in_Bottle_ml >= "Global_DB".Other_Parameters.Liquid_B_pct;
END_REGION
END_ORGANIZATION_BLOCK

FUNCTION "Filling_Logik" : Void   // FC5, LAD
{ S7_Optimized_Access := 'TRUE' }
VERSION : 0.1
// stored: AutoNumber true, IsIECCheckEnabled false, SetENOAutomatically false, UDAEnableTagReadback false
   VAR_INPUT
      PS2_Filling_Station : Bool;
      FIC_B102 : Int;
      Liquid_AorB_in_Bottle_ml : Real;
      Liquid_AorB_pct : Int;
      Wait_to_fill : Time;
   END_VAR
   VAR_OUTPUT
      Flow_ml_per_sec : Real;
      FillingData_LiqAorB_ml : Real;
   END_VAR
   VAR_IN_OUT
      Outlet_of_tanks : Bool;
   END_VAR
   VAR_TEMP
      PTRIG1 : Bool;
      PTRIG2 : Bool;
      PTRIG3 : Bool;
      PTRIG4 : Bool;
   END_VAR
BEGIN

REGION Network 1
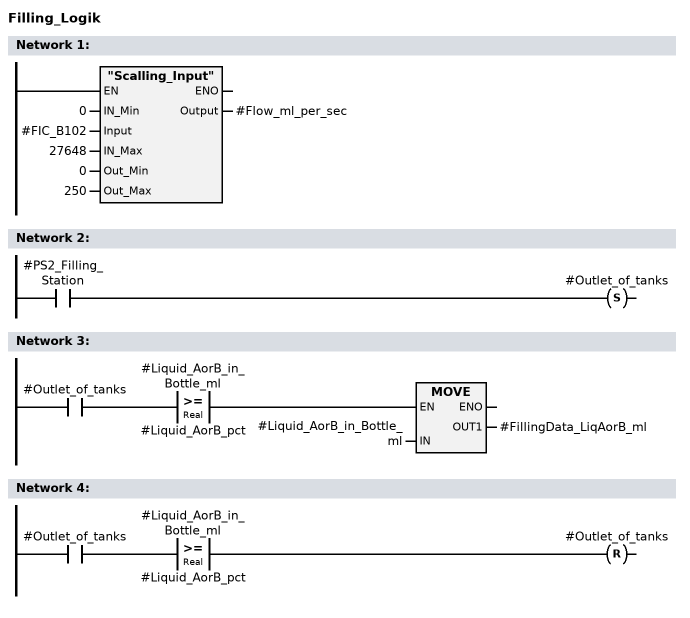
   RUNG wire#powerrail
      "Scalling_Input"(IN_Min := 0, Input := #FIC_B102, IN_Max := 27648, Out_Min := 0, Out_Max := 250, Output => #Flow_ml_per_sec)
   END_RUNG
   // the same network as SCL:
   "Scalling_Input"(IN_Min := 0,
                    Input := #FIC_B102,
                    IN_Max := 27648,
                    Out_Min := 0,
                    Out_Max := 250,
                    Output => #Flow_ml_per_sec);
END_REGION

REGION Network 2
   RUNG wire#powerrail
      Contact( #PS2_Filling_Station )
      S_Coil( #Outlet_of_tanks )
   END_RUNG
   // the same network as SCL:
   IF #PS2_Filling_Station THEN #Outlet_of_tanks := TRUE; END_IF;
END_REGION

REGION Network 3
   RUNG wire#powerrail
      Contact( #Outlet_of_tanks )
      { S7_Templates := "SrcType := Real" } GE_Contact(in1 := #Liquid_AorB_in_Bottle_ml, in2 := #Liquid_AorB_pct)
      Move(in := #Liquid_AorB_in_Bottle_ml, out1 => #FillingData_LiqAorB_ml)
   END_RUNG
   // the same network as SCL:
   IF #Outlet_of_tanks AND (#Liquid_AorB_in_Bottle_ml >= #Liquid_AorB_pct) THEN
       #FillingData_LiqAorB_ml := #Liquid_AorB_in_Bottle_ml;
   END_IF;
END_REGION

REGION Network 4
   RUNG wire#powerrail
      Contact( #Outlet_of_tanks )
      { S7_Templates := "SrcType := Real" } GE_Contact(in1 := #Liquid_AorB_in_Bottle_ml, in2 := #Liquid_AorB_pct)
      R_Coil( #Outlet_of_tanks )
   END_RUNG
   // the same network as SCL:
   IF #Outlet_of_tanks AND (#Liquid_AorB_in_Bottle_ml >= #Liquid_AorB_pct) THEN
       #Outlet_of_tanks := FALSE;
   END_IF;
END_REGION
END_FUNCTION

FUNCTION_BLOCK "Filling_Logic"   // FB2, LAD
{ S7_Optimized_Access := 'TRUE' }
VERSION : 0.1
// stored: AutoNumber true, IsIECCheckEnabled false, IsRetainMemResEnabled false, MemoryReserve 100, SetENOAutomatically false, UDAEnableTagReadback false
   VAR_INPUT
      PS2_Filling_Station : Bool;
      FIC_B102 : Int;
      Liquid_AorB_in_Bottle_ml : Real;
      Liquid_AorB_pct : Int;
      PTRIG3 : Bool;
      PTRIG2 : Bool;
      Wait_to_fill : Time;
   END_VAR
   VAR_OUTPUT
      Outlet_of_tanks : Bool;
      Flow_ml_per_sec : Real;
      PTRIG1 : Bool;
      FillingData_LiqAorB_ml : Real;
   END_VAR
BEGIN

REGION Network 1
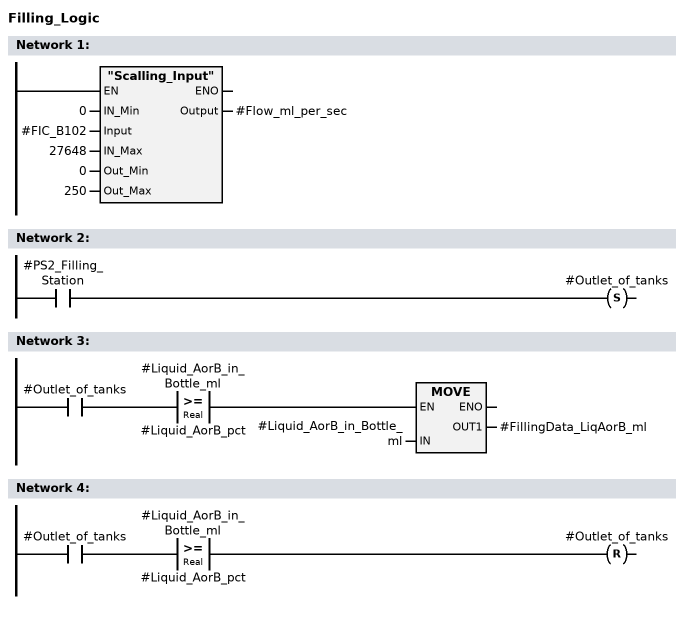
   RUNG wire#powerrail
      "Scalling_Input"(IN_Min := 0, Input := #FIC_B102, IN_Max := 27648, Out_Min := 0, Out_Max := 250, Output => #Flow_ml_per_sec)
   END_RUNG
   // the same network as SCL:
   "Scalling_Input"(IN_Min := 0,
                    Input := #FIC_B102,
                    IN_Max := 27648,
                    Out_Min := 0,
                    Out_Max := 250,
                    Output => #Flow_ml_per_sec);
END_REGION

REGION Network 2
   RUNG wire#powerrail
      Contact( #PS2_Filling_Station )
      S_Coil( #Outlet_of_tanks )
   END_RUNG
   // the same network as SCL:
   IF #PS2_Filling_Station THEN #Outlet_of_tanks := TRUE; END_IF;
END_REGION

REGION Network 3
   RUNG wire#powerrail
      Contact( #Outlet_of_tanks )
      { S7_Templates := "SrcType := Real" } GE_Contact(in1 := #Liquid_AorB_in_Bottle_ml, in2 := #Liquid_AorB_pct)
      Move(in := #Liquid_AorB_in_Bottle_ml, out1 => #FillingData_LiqAorB_ml)
   END_RUNG
   // the same network as SCL:
   IF #Outlet_of_tanks AND (#Liquid_AorB_in_Bottle_ml >= #Liquid_AorB_pct) THEN
       #FillingData_LiqAorB_ml := #Liquid_AorB_in_Bottle_ml;
   END_IF;
END_REGION

REGION Network 4
   RUNG wire#powerrail
      Contact( #Outlet_of_tanks )
      { S7_Templates := "SrcType := Real" } GE_Contact(in1 := #Liquid_AorB_in_Bottle_ml, in2 := #Liquid_AorB_pct)
      R_Coil( #Outlet_of_tanks )
   END_RUNG
   // the same network as SCL:
   IF #Outlet_of_tanks AND (#Liquid_AorB_in_Bottle_ml >= #Liquid_AorB_pct) THEN
       #Outlet_of_tanks := FALSE;
   END_IF;
END_REGION
END_FUNCTION_BLOCK

FUNCTION "Scalling_Output" : Void   // FC2, FBD
{ S7_Optimized_Access := 'TRUE' }
VERSION : 0.1
// stored: AutoNumber true, IsIECCheckEnabled false, SetENOAutomatically false, UDAEnableTagReadback false
   VAR_INPUT
      IN_Min : Int;
      Input : Int;
      IN_Max : Int;
      Out_Min : Int;
      Out_Max : Int;
   END_VAR
   VAR_OUTPUT
      Output : Int;
   END_VAR
   VAR_TEMP
      Normed : Real;
   END_VAR
BEGIN

REGION Network 1
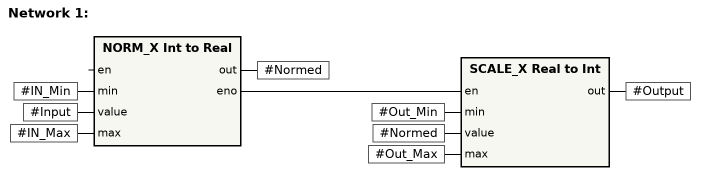
   #Normed := NORM_X(MIN := #IN_Min, VALUE := #Input, MAX := #IN_Max);
   #Output := SCALE_X(MIN := #Out_Min, VALUE := #Normed, MAX := #Out_Max);
END_REGION
END_FUNCTION

DATA_BLOCK "ProductionData_Reset_DB"   // DB13
VERSION : 0.1
// stored: AutoNumber true, DBAccessibleFromOPCUA true, InstanceOfName ProductionData_Reset, InstanceOfType FB
"ProductionData_Reset"
BEGIN
END_DATA_BLOCK

DATA_BLOCK "Alarm_Logic_DB"   // DB7
VERSION : 0.1
// stored: AutoNumber true, DBAccessibleFromOPCUA true, InstanceOfName Alarm_Logic, InstanceOfType FB
"Alarm_Logic"
BEGIN
END_DATA_BLOCK

DATA_BLOCK "Filling_Logic_DB"   // DB4
VERSION : 0.1
// stored: AutoNumber true, DBAccessibleFromOPCUA true, InstanceOfName Filling_Logic, InstanceOfType FB
"Filling_Logic"
BEGIN
END_DATA_BLOCK

DATA_BLOCK "Filling_Logic_DB_1"   // DB5
VERSION : 0.1
// stored: AutoNumber true, DBAccessibleFromOPCUA true, InstanceOfName Filling_Logic, InstanceOfType FB
"Filling_Logic"
BEGIN
END_DATA_BLOCK

DATA_BLOCK "Operation_cycle_DB"   // DB15
VERSION : 0.1
// stored: AutoNumber true, DBAccessibleFromOPCUA true, InstanceOfName Operation_cycle, InstanceOfType FB
"Operation_cycle"
BEGIN
END_DATA_BLOCK

DATA_BLOCK "Re-filling_Logic_DB"   // DB2
VERSION : 0.1
// stored: AutoNumber true, DBAccessibleFromOPCUA true, InstanceOfName Re-filling_Logic, InstanceOfType FB
"Re-filling_Logic"
BEGIN
END_DATA_BLOCK

DATA_BLOCK "Tank1_DB"   // DB9
VERSION : 0.1
// stored: AutoNumber true, DBAccessibleFromOPCUA true, InstanceOfName Tank1, InstanceOfType FB
"Tank1"
BEGIN
END_DATA_BLOCK

DATA_BLOCK "Tank2_DB"   // DB10
VERSION : 0.1
// stored: AutoNumber true, DBAccessibleFromOPCUA true, InstanceOfName Tank2, InstanceOfType FB
"Tank2"
BEGIN
END_DATA_BLOCK

DATA_BLOCK "Cycle_time"   // DB14
{ S7_Optimized_Access := 'TRUE' }
// stored: AutoNumber true, DBAccessibleFromOPCUA true, InstanceOfName IEC_TIMER, OfSystemLibElement IEC_TIMER, OfSystemLibVersion 1.0
"IEC_TIMER"
   // VAR
   //    PT : Time;
   //    ET { ExternalWritable := 'False'} : Time;
   //    IN : Bool;
   //    Q { ExternalWritable := 'False'} : Bool;
   // END_VAR
BEGIN
END_DATA_BLOCK

DATA_BLOCK "IEC_Timer_0_DB_1"   // DB6
{ S7_Optimized_Access := 'TRUE' }
// stored: AutoNumber true, DBAccessibleFromOPCUA true, InstanceOfName IEC_TIMER, OfSystemLibElement IEC_TIMER, OfSystemLibVersion 1.0
"IEC_TIMER"
   // VAR
   //    PT : Time;
   //    ET { ExternalWritable := 'False'} : Time;
   //    IN : Bool;
   //    Q { ExternalWritable := 'False'} : Bool;
   // END_VAR
BEGIN
END_DATA_BLOCK

DATA_BLOCK "IEC_Timer_0_DB_7"   // DB11
{ S7_Optimized_Access := 'TRUE' }
// stored: AutoNumber true, DBAccessibleFromOPCUA true, InstanceOfName IEC_TIMER, OfSystemLibElement IEC_TIMER, OfSystemLibVersion 1.0
"IEC_TIMER"
   // VAR
   //    PT : Time;
   //    ET { ExternalWritable := 'False'} : Time;
   //    IN : Bool;
   //    Q { ExternalWritable := 'False'} : Bool;
   // END_VAR
BEGIN
END_DATA_BLOCK

DATA_BLOCK "IEC_Timer_0_DB_999"   // DB8
{ S7_Optimized_Access := 'TRUE' }
// stored: AutoNumber true, DBAccessibleFromOPCUA true, InstanceOfName IEC_TIMER, OfSystemLibElement IEC_TIMER, OfSystemLibVersion 1.0
"IEC_TIMER"
   // VAR
   //    PT : Time;
   //    ET { ExternalWritable := 'False'} : Time;
   //    IN : Bool;
   //    Q { ExternalWritable := 'False'} : Bool;
   // END_VAR
BEGIN
END_DATA_BLOCK

DATA_BLOCK "IEC_Timer_6_DB_1"   // DB3
{ S7_Optimized_Access := 'TRUE' }
// stored: AutoNumber true, DBAccessibleFromOPCUA true, InstanceOfName IEC_TIMER, OfSystemLibElement IEC_TIMER, OfSystemLibVersion 1.0
"IEC_TIMER"
   // VAR
   //    PT : Time;
   //    ET { ExternalWritable := 'False'} : Time;
   //    IN : Bool;
   //    Q { ExternalWritable := 'False'} : Bool;
   // END_VAR
BEGIN
END_DATA_BLOCK
